// TIA Portal project "Project1" (V15)

(* hardware
DEVICE "S7-1200 station_1"  S7-1200 Station
   slot 0: "Rack_0"  S7-1200 Rack  Rack  V1.0
   slot 1: "PLC_1"  CPU 1214C DC/DC/DC  6ES7 214-1AG40-0XB0  V4.2
*)

// ===== PLC "PLC_1"  CPU 1214C DC/DC/DC =====

VAR_GLOBAL   // PLC tag table "Default tag table"
   "Tag_1" AT %I0.1 : Bool;
   "Tag_2" AT %Q0.0 : Bool;
   "Tag_3" AT %M0.0 : Bool;
END_VAR

ORGANIZATION_BLOCK "Main"   // OB1, LAD, ProgramCycle
TITLE = "Main Program Sweep (Cycle)"
{ S7_Optimized_Access := 'TRUE' }
VERSION : 0.1
   VAR_INPUT
      Initial_Call : Bool;   // Initial call of this OB
      Remanence : Bool;   // =True, if remanent data are available
   END_VAR
   VAR_TEMP   // added for the SCL form of the ladder/FBD networks
      _w1 : Bool;
      _w2 : Bool;
   END_VAR
BEGIN

REGION Network 1
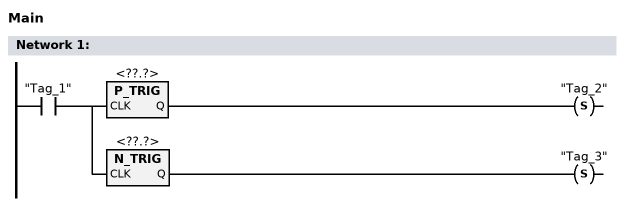
   RUNG wire#powerrail
      Contact( "Tag_1" )
      wire#w1
      P_Trig(  )
      S_Coil( "Tag_2" )
   END_RUNG
   RUNG wire#w1
      N_Trig(  )
      S_Coil( "Tag_3" )
   END_RUNG
   // the same network as SCL:
   #_w1 := "Tag_1" AND NOT <??.?>;   // rising edge
   <??.?> := "Tag_1";
   IF #_w1 THEN "Tag_2" := TRUE; END_IF;
   #_w2 := NOT "Tag_1" AND <??.?>;   // falling edge
   <??.?> := "Tag_1";
   IF #_w2 THEN "Tag_3" := TRUE; END_IF;
END_REGION
END_ORGANIZATION_BLOCK